FUNCTION_BLOCK OnLinkedListChangedHandler IMPLEMENTS I_EventHandler
VAR
	expectedOriginator : I_LinkedList;
	_eventReceived : BOOL;
	fromExpected : BOOL;
END_VAR

PROPERTY PUBLIC EventReceived : BOOL
GET
EventReceived := _eventReceived;
END_GET
END_PROPERTY

METHOD FB_init : BOOL
VAR_INPUT
	bInitRetains : BOOL; // if TRUE, the retain variables are initialized (warm start / cold start)
	bInCopyCode : BOOL;  // if TRUE, the instance afterwards gets moved into the copy code (online change)
	ExpectedOriginator : I_LinkedList;
END_VAR
SetExpectedOriginator(ExpectedOriginator);
END_METHOD

PROPERTY PUBLIC FromExpectedOriginator : BOOL
GET
FromExpectedOriginator := fromExpected;
END_GET
END_PROPERTY

METHOD PUBLIC HandleEvent
VAR_INPUT
	Event : I_Event;
END_VAR
VAR
	linkedListChangedEvent : I_LinkedListChangedEvent;
END_VAR
IF __QUERYINTERFACE(Event, linkedListChangedEvent) THEN
	_eventReceived := TRUE;
	fromExpected := linkedListChangedEvent.TargetLinkedList = expectedOriginator;
END_IF
END_METHOD

METHOD PUBLIC Reset
VAR_INPUT
END_VAR
_eventReceived := FALSE;
fromExpected := FALSE;
END_METHOD

METHOD PUBLIC SetExpectedOriginator
VAR_INPUT
	ExpectedOriginator : I_LinkedList;
END_VAR
this^.expectedOriginator := ExpectedOriginator;
END_METHOD

END_FUNCTION_BLOCK

(* stored: Version 1.1.0.1, ProductVersion 3.1.4024.12
   POU OnLinkedListChangedHandler: Id {624d4e7f-4cae-4871-b4f1-8321a9ffcc81}, SpecialFunc None
   Folder Constructor: Id {ec17492d-00d9-4fd5-b491-0cd3eba4e243}
   Property EventReceived: Id {0c5b5b1e-ae6f-47f5-a0eb-647efc7c77b6}
   Get Get: Id {ae6a466a-a62e-42cb-a47e-fd1f687ce1c6}
   Method FB_init: Id {faf05151-4d3d-4158-a290-ad0b87a7a5c3}
   Property FromExpectedOriginator: Id {4115df43-c1b3-41a9-8397-99718f881682}
   Get Get: Id {39f84cde-518a-44ee-8c03-548ffc38dd3b}
   Method HandleEvent: Id {d6b42d48-9627-422d-af26-eee80c59dc1d}
   Method Reset: Id {2e6c2f99-e06e-4d4a-8d59-448660c53c36}
   Method SetExpectedOriginator: Id {81554e37-adf6-4986-bdd7-b49945ba620a} *)
